// TIA Portal V20 export
FUNCTION_BLOCK "FB_Blowing"   // FB63, SCL
{ S7_Optimized_Access := 'TRUE' }
// stored: AutoNumber false, MemoryReserve 100, SetENOAutomatically false
   VAR_INPUT
      iStartSeqCond : Bool;   // Start Sequence Conditions
      iJobReq : Bool;   // Job Request - From Main
      iShuttleBlowingPos : Bool;   // Load/Unload Pos. Reached - Param
      iShuttleBlowingPosSetPoint : LReal;   // Load/Unload Pos. Setpoint - Param
      iAxisV_BlowingPos : Bool;
      iAxisV_BlowingPosSetPoint : LReal;
      iAxisW_SafePos : Bool;
      iAxisW_SafePosSetPoint : LReal;
      iAxisW_BlowingPos : Bool;
      iAxisW_BlowingPosSetPoint : LReal;
      iShuttleMoving : Bool;   // Shuttle is moving - From FB_LoaderAxis
      iShuttleInPos : Bool;   // Shuttle pos. reached - From FB_LoaderAxis
      iAxisV_Moving : Bool;   // Shuttle is moving
      iAxisV_InPos : Bool;
      iAxisW_Moving { ExternalAccessible := 'False'; ExternalVisible := 'False'; ExternalWritable := 'False'} : Bool;   // Shuttle is moving
      iAxisW_InPos : Bool;
      iBlowingTime : Time;
      iPLC_DateAndTime : DTL;
      iStepPause : Bool;
   END_VAR
   VAR_OUTPUT
      oShuttleStartReq { ExternalAccessible := 'False'; ExternalVisible := 'False'; ExternalWritable := 'False'} : Bool;   // Shuttle Start Order - To FB_LoaderAxis
      oShuttlePosSetPoint { ExternalAccessible := 'False'; ExternalVisible := 'False'; ExternalWritable := 'False'} : Real;   // Shuttle Position Setpoint - To FB_LoaderAxis
      oAxisV_StartReq : Bool;
      oAxisV_PosSetPoint : Real;
      oAxisW_StartReq : Bool;
      oAxisW_PosSetPoint : Real;
      oBlowingReq : Bool;
   END_VAR
   VAR
      sCurrent_Step_NB : Int;   // Active Step Number
      sCheck_Step_Condition : Bool;
      sOneStepForward : Bool;
      sRTOneStepForward : R_TRIG;
      sOneStepMode { S7_SetPoint := 'True'} : Bool;
      sStepForward : Bool;
      sInterface : "UDT_SequenceInterface";
      sShuttleStartReq { ExternalAccessible := 'False'; ExternalVisible := 'False'; ExternalWritable := 'False'} : Bool;
      sShuttlePosSetPoint { ExternalAccessible := 'False'; ExternalVisible := 'False'; ExternalWritable := 'False'} : Real;
      sAxisV_StartReq : Bool;
      sAxisV_PosSetPoint : Real;
      sAxisW_StartReq : Bool;
      sAxisW_PosSetPoint : Real;
      sBlowingReq : Bool;   // Drilled Part To Unload - From FB_Position
      sBlowingTimerStart : Bool;
      sBlowingTimer : TP_TIME;
      sFT_BlowingTimer { S7_SetPoint := 'True'} : F_TRIG;
      sHistory : Struct
         Activation : Bool;
         Steps : Array[0..99] of Int;
         Date_Time : Array[0..99] of DTL;
      END_STRUCT;
      StepText : "FB_GetTextErrorCode";
   END_VAR
   VAR_TEMP
      tIndex : Int;   // Index
   END_VAR
   VAR CONSTANT
      S00_INIT : Int := 0;
      S10_CHECK_BLOWING_OPTION : Int := 10;
      S20_SHUTTLE_TO_BLOWING_POS_START_REQ : Int := 20;
      S30_SHUTTLE_TO_BLOWING_POS_REACHED : Int := 30;
      S40_AXIS_W_TO_SAFE_POS_START_REQ : Int := 40;
      S50_AXIS_W_TO_SAFE_POS_REACHED : Int := 50;
      S60_AXIS_V_TO_BLOWING_POS_START_REQ : Int := 60;
      S70_AXIS_V_TO_BLOWING_POS_REACHED : Int := 70;
      S80_AXIS_W_TO_BLOWING_POS_START_REQ : Int := 80;
      S90_AXIS_W_TO_BLOWING_POS_REACHED : Int := 90;
      S100_BLOWING_TIMER_START_REQ : Int := 100;
      S195_JOB_DONE : Int := 195;
   END_VAR
   // StepText.sCode_error[0].ErrorCode := 0;
   // StepText.sCode_error[1].ErrorCode := 10;
   // StepText.sCode_error[2].ErrorCode := 20;
   // StepText.sCode_error[3].ErrorCode := 30;
   // StepText.sCode_error[4].ErrorCode := 40;
   // StepText.sCode_error[5].ErrorCode := 50;
   // StepText.sCode_error[6].ErrorCode := 60;
   // StepText.sCode_error[7].ErrorCode := 70;
   // StepText.sCode_error[8].ErrorCode := 80;
   // StepText.sCode_error[9].ErrorCode := 90;
   // StepText.sCode_error[10].ErrorCode := 95;
BEGIN
   REGION Description header 
       //==================================================================================
       // POSALUX Swiss SA / (C) Copyright 2025
       //----------------------------------------------------------------------------------
       // Title: FB_Blowing
       // Comment/Function: 
       // Author: Fabien WALDT
       // Engineering: TIA Portal v17
       //----------------------------------------------------------------------------------
       // Change log table:
       // Version  | Date     | Expert in charge | Changes applied
       // ---------|----------|------------------|-----------------------------------------
       // 00.00.01 | 20250527 | WFA              | First released version
       // =================================================================================
   END_REGION

   REGION Define condition to start
       IF #iStartSeqCond THEN
           #sInterface.SequenceReleased := TRUE;
       ELSE
           // Standard sequencer controls
           #sInterface.SequenceReleased := FALSE;
           #sCurrent_Step_NB := #S00_INIT;
           #sInterface.SequenceRun := FALSE;
           #sInterface.JobDone := FALSE;
           #sCheck_Step_Condition := FALSE;

           // Dedicated sequencer controls
           #sShuttleStartReq := FALSE;
           #sShuttlePosSetPoint := 0.0;
           #sAxisV_StartReq := FALSE;
           #sAxisV_PosSetPoint := 0.0;
           #sAxisW_StartReq := FALSE;
           #sAxisW_PosSetPoint := 0.0;
           #sBlowingReq := FALSE;
           #sBlowingTimerStart := FALSE;

           // Add specifics controls 
       END_IF;

       // Reset interface error
       IF #sInterface.Reset THEN
           #sInterface.Error := FALSE;
       END_IF;

       // Reset start when axis in position
       IF #iShuttleInPos THEN
           #sShuttleStartReq := FALSE;
       END_IF;
       IF #iAxisV_InPos THEN
           #sAxisV_StartReq := FALSE;
       END_IF;
       IF #iAxisW_InPos THEN
           #sAxisW_StartReq := FALSE;
       END_IF;

       // One step forward
       #sRTOneStepForward.CLK := #sOneStepForward;
       #sRTOneStepForward();
       #sStepForward := (NOT #sOneStepMode OR (#sOneStepMode AND #sRTOneStepForward.Q)) AND NOT #iStepPause;
       #sOneStepForward := FALSE;

       // Action only true in dedicated steps
       #sBlowingReq := FALSE;

       // Blowing Timer
       #sBlowingTimer(IN := #sBlowingTimerStart AND #sStepForward,
                      PT := #iBlowingTime);

       #sFT_BlowingTimer(CLK := #sBlowingTimer.Q);

       #sBlowingReq := #sBlowingTimer.Q;
   END_REGION

   REGION Sequence Function
       CASE #sCurrent_Step_NB OF
           #S00_INIT:
               REGION S00 INIT
                   #sCheck_Step_Condition := TRUE;
               END_REGION
           #S10_CHECK_BLOWING_OPTION:
               REGION S10_CHECK_BLOWING_OPTION
                   #sCheck_Step_Condition := TRUE;
               END_REGION
           #S20_SHUTTLE_TO_BLOWING_POS_START_REQ:
               REGION S20_SHUTTLE_TO_BLOWING_POS_START_REQ
                   #sShuttleStartReq := NOT #iShuttleBlowingPos;
                   #sShuttlePosSetPoint := LREAL_TO_REAL(#iShuttleBlowingPosSetPoint);
                   #sCheck_Step_Condition := TRUE;
               END_REGION
           #S30_SHUTTLE_TO_BLOWING_POS_REACHED:
               REGION S30_SHUTTLE_TO_BLOWING_POS_REACHED
                   #sCheck_Step_Condition := TRUE;
               END_REGION
           #S40_AXIS_W_TO_SAFE_POS_START_REQ:
               REGION S40_AXIS_W_TO_SAFE_POS_START_REQ
                   #sAxisW_StartReq := NOT #iAxisW_SafePos;
                   #sAxisW_PosSetPoint := LREAL_TO_REAL(#iAxisW_SafePosSetPoint);
                   #sCheck_Step_Condition := TRUE;
               END_REGION
           #S50_AXIS_W_TO_SAFE_POS_REACHED:
               REGION S50_AXIS_W_TO_SAFE_POS_REACHED
                   #sCheck_Step_Condition := TRUE;
               END_REGION
           #S60_AXIS_V_TO_BLOWING_POS_START_REQ:
               REGION S60_AXIS_V_TO_BLOWING_POS_START_REQ
                   #sAxisV_StartReq := NOT #iAxisV_BlowingPos;
                   #sAxisV_PosSetPoint := LREAL_TO_REAL(#iAxisV_BlowingPosSetPoint);
                   #sCheck_Step_Condition := TRUE;
               END_REGION
           #S70_AXIS_V_TO_BLOWING_POS_REACHED:
               REGION S70_AXIS_V_TO_BLOWING_POS_REACHED
                   #sCheck_Step_Condition := TRUE;
               END_REGION
           #S80_AXIS_W_TO_BLOWING_POS_START_REQ:
               REGION S80_AXIS_W_TO_BLOWING_POS_START_REQ
                   #sAxisW_StartReq := NOT #iAxisW_BlowingPos;
                   #sAxisW_PosSetPoint := LREAL_TO_REAL(#iAxisW_BlowingPosSetPoint);
                   #sCheck_Step_Condition := TRUE;
               END_REGION
           #S90_AXIS_W_TO_BLOWING_POS_REACHED:
               REGION S90_AXIS_W_TO_BLOWING_POS_REACHED
                   #sCheck_Step_Condition := TRUE;
               END_REGION
           #S100_BLOWING_TIMER_START_REQ:
               REGION S100_BLOWING TIMER_START_REQ
                   #sBlowingTimerStart := TRUE;
                   #sCheck_Step_Condition := TRUE;
               END_REGION
           #S195_JOB_DONE:
               REGION S195_JOB_DONE
                   #sBlowingTimerStart := FALSE;
                   #sInterface.JobDone := TRUE;
                   #sCheck_Step_Condition := TRUE;
               END_REGION
           ELSE:
               #sInterface.Error := TRUE;
       END_CASE;
   END_REGION

   REGION Sequence Next Step Condition
       IF #sCheck_Step_Condition THEN
           CASE #sCurrent_Step_NB OF
               #S00_INIT:
                   REGION S00 INIT
                       IF #sInterface.SequenceReleased AND #iJobReq THEN
                           #sCurrent_Step_NB := #S10_CHECK_BLOWING_OPTION;
                           #sInterface.SequenceRun := TRUE;
                           #sCheck_Step_Condition := FALSE;
                       ELSE
                           #sInterface.SequenceRun := FALSE;
                       END_IF;
                   END_REGION
               #S10_CHECK_BLOWING_OPTION:
                   REGION S10_CHECK_BLOWING_OPTION
                       IF #sInterface.SequenceReleased AND #sStepForward AND "DB_LoaderOptions".Blowing.Inside AND NOT "DB_LoaderOptions".Blowing.Disabled  THEN
                           #sCurrent_Step_NB := #S20_SHUTTLE_TO_BLOWING_POS_START_REQ;
                           #sCheck_Step_Condition := FALSE;
                       ELSIF #sInterface.SequenceReleased AND #sStepForward AND (NOT "DB_LoaderOptions".Blowing.Inside OR NOT "DB_LoaderOptions".Blowing.Disabled)  THEN
                           #sCurrent_Step_NB := #S195_JOB_DONE;
                           #sCheck_Step_Condition := FALSE;
                       END_IF;
                   END_REGION
               #S20_SHUTTLE_TO_BLOWING_POS_START_REQ:
                   REGION S20_SHUTTLE_TO_BLOWING_POS_START_REQ
                       IF #sInterface.SequenceReleased AND (#iShuttleMoving OR #iShuttleBlowingPos) THEN
                           #sCurrent_Step_NB := #S30_SHUTTLE_TO_BLOWING_POS_REACHED;
                           #sCheck_Step_Condition := FALSE;
                       END_IF;
                   END_REGION
               #S30_SHUTTLE_TO_BLOWING_POS_REACHED:
                   REGION S30_SHUTTLE_TO_BLOWING_POS_REACHED
                       IF #sInterface.SequenceReleased AND #sStepForward AND NOT #sShuttleStartReq AND #iShuttleBlowingPos THEN
                           #sCurrent_Step_NB := #S40_AXIS_W_TO_SAFE_POS_START_REQ;
                           #sCheck_Step_Condition := FALSE;
                       END_IF;
                   END_REGION
               #S40_AXIS_W_TO_SAFE_POS_START_REQ:
                   REGION S40_AXIS_W_TO_SAFE_POS_START_REQ
                       IF #sInterface.SequenceReleased AND (#iAxisW_Moving OR #iAxisW_SafePos) THEN
                           #sCurrent_Step_NB := #S50_AXIS_W_TO_SAFE_POS_REACHED;
                           #sCheck_Step_Condition := FALSE;
                       END_IF;
                   END_REGION
               #S50_AXIS_W_TO_SAFE_POS_REACHED:
                   REGION S50_AXIS_W_TO_SAFE_POS_REACHED
                       IF #sInterface.SequenceReleased AND #sStepForward AND NOT #sAxisW_StartReq AND #iAxisW_SafePos THEN
                           #sCurrent_Step_NB := #S60_AXIS_V_TO_BLOWING_POS_START_REQ;
                           #sCheck_Step_Condition := FALSE;
                       END_IF;
                   END_REGION
               #S60_AXIS_V_TO_BLOWING_POS_START_REQ:
                   REGION S60_AXIS_V_TO_BLOWING_POS_START_REQ
                       IF #sInterface.SequenceReleased AND #sStepForward AND (#iAxisV_Moving OR #iAxisV_BlowingPos) THEN
                           #sCurrent_Step_NB := #S70_AXIS_V_TO_BLOWING_POS_REACHED;
                           #sCheck_Step_Condition := FALSE;
                       END_IF;
                   END_REGION
               #S70_AXIS_V_TO_BLOWING_POS_REACHED:
                   REGION S70_AXIS_V_TO_BLOWING_POS_REACHED
                       IF #sInterface.SequenceReleased AND #sStepForward AND NOT #sAxisV_StartReq AND #iAxisV_BlowingPos THEN
                           #sCurrent_Step_NB := #S80_AXIS_W_TO_BLOWING_POS_START_REQ;
                           #sCheck_Step_Condition := FALSE;
                       END_IF;
                   END_REGION
               #S80_AXIS_W_TO_BLOWING_POS_START_REQ:
                   REGION S80_AXIS_W_TO_BLOWING_POS_START_REQ
                       IF #sInterface.SequenceReleased AND (#iAxisW_Moving OR #iAxisW_BlowingPos) THEN
                           #sCurrent_Step_NB := #S90_AXIS_W_TO_BLOWING_POS_REACHED;
                           #sCheck_Step_Condition := FALSE;
                       END_IF;
                   END_REGION
               #S90_AXIS_W_TO_BLOWING_POS_REACHED:
                   REGION S90_AXIS_W_TO_BLOWING_POS_REACHED
                       IF #sInterface.SequenceReleased AND #sStepForward AND NOT #sAxisW_StartReq AND #iAxisW_BlowingPos THEN
                           #sCurrent_Step_NB := #S100_BLOWING_TIMER_START_REQ;
                           #sCheck_Step_Condition := FALSE;
                       END_IF;
                   END_REGION
               #S100_BLOWING_TIMER_START_REQ:
                   REGION S100_BLOWING_TIMER_START_REQ
                       IF #sInterface.SequenceReleased AND #sStepForward AND #sFT_BlowingTimer.Q THEN
                           #sCurrent_Step_NB := #S195_JOB_DONE;
                           #sCheck_Step_Condition := FALSE;
                       END_IF;
                   END_REGION
               #S195_JOB_DONE:
                   REGION S95_JOB_DONE
                       IF NOT #iJobReq THEN
                           #sCurrent_Step_NB := #S00_INIT;
                           #sCheck_Step_Condition := FALSE;
                           #sInterface.JobDone := FALSE;
                       END_IF;
                   END_REGION
               ELSE
                   #sInterface.Error := TRUE;
           END_CASE;
       END_IF;
   END_REGION

   REGION Outputs Update
       #oShuttleStartReq := #sShuttleStartReq;
       #oShuttlePosSetPoint := #sShuttlePosSetPoint;
       #oAxisV_StartReq := #sAxisV_StartReq;
       #oAxisV_PosSetPoint := #sAxisV_PosSetPoint;
       #oAxisW_StartReq := #sAxisW_StartReq;
       #oAxisW_PosSetPoint := #sAxisW_PosSetPoint;
       #oBlowingReq := #sBlowingReq;
   END_REGION

   REGION Steps - Date and Time History
       IF #sHistory.Activation THEN
           IF #sHistory.Steps[0] <> #sCurrent_Step_NB THEN
               FOR #tIndex := 98 TO 0 BY -1 DO
                   #sHistory.Steps[#tIndex + 1] := #sHistory.Steps[#tIndex];
                   #sHistory.Date_Time[#tIndex + 1] := #sHistory.Date_Time[#tIndex];
               END_FOR;
               #sHistory.Steps[0] := #sCurrent_Step_NB;
               #sHistory.Date_Time[0] := #iPLC_DateAndTime;
           END_IF;
       END_IF;
   END_REGION

   REGION Steps Text
       #StepText(iErrorCode := #sCurrent_Step_NB,
                 oErrorText => #StepText.oErrorText);
   END_REGION
END_FUNCTION_BLOCK
